PROGRAM MAIN
VAR
	T :							REAL := 0.001;	
	K :							REAL := 10;
	PID_Parameter :				PID_Parameter_Strukt;
	Modus :						System_Modus_Enum := System_Modus_Enum.System_Init;
	PID_1 :						PID_Regler;
	
	r0 :						REAL := 0;	//Goal RPM
	dc_Encoder :				UINT := 0;	//DC Encoder Impulses (0-65536)
	dc_Encoder_old :			UINT := 0;
	dc_OverflowBit :			BOOL := 0;	//DC Encoder Overflow 
	dc_UnderflowBit :			BOOL := 0;	//DC Encoder Underflow
	dc_RPM : 					REAL := 0;	//DC Motor RPM (1 Rotation = 32,768 Impulses)
	
	
	e0 :						REAL := 0;
END_VAR
//

CASE Modus OF
	System_Modus_Enum.System_Init:
	PID_Parameter.Kp := 100/K;
	PID_Parameter.Ti := 1;
	PID_Parameter.Td := 2;
	PID_Parameter.N := 10;
	PID_Parameter.umax := 10;
	PID_Parameter.umin := 0;
	PID_Parameter.ARW := TRUE;
	PID_Parameter.Tr := 0.1;
	Modus := System_Modus_Enum.System_Run
	;
	System_Modus_Enum.System_Run:
	dc_RPM := dc_Encoder - dc_Encoder_old;
	e0 := r0;
	PID_1(r1 := r0, y1 := 0, Modus := Modus, Param := PID_Parameter, T := T);
	dc_Encoder_old := dc_Encoder;
	;
END_CASE

END_PROGRAM

(* stored: Version 1.1.0.1, ProductVersion 3.1.4024.13
   POU MAIN: Id {ec08e590-4119-4f47-b80e-690b31a799d1}, SpecialFunc None *)
